SYSTEM Test_6 (* System Configuration *)
  (* Standard: 61499-1 *)
  (* Version 0.3, 2003-12-05, JHC, Rockwell Automation, Renamed from NEWSYSTEM. *)
  (* Version 0.2, 2002-11-05, JHC, Rockwell Automation, Fixed missing (empty) FBD in Application. *)
  (* Version 0.1, 2002-01-17, JHC, Rockwell Automation, Minor cleanup *)
  (* Version 0.0, 2000-05-27, JHC, Rockwell Automation *)
  APPLICATION APP1
  END_APPLICATION
  DEVICE DEV1 : FRAME_DEVICE(BOUNDS := [110,110,300,300], GRID := [1,1])
    RESOURCE RES1 : PANEL_RESOURCE(ROWS := 2, COLS := 2)
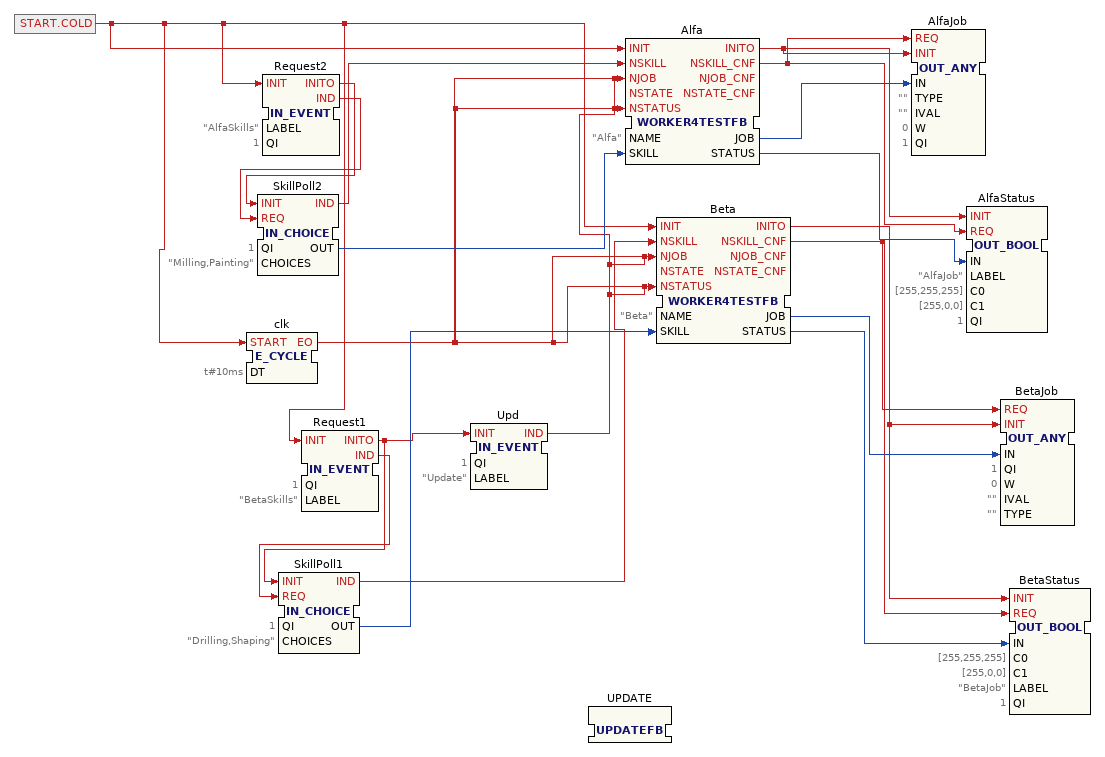
      FBS
        Alfa : WORKER4TESTFB(NAME := "Alfa");
        Beta : WORKER4TESTFB(NAME := "Beta");
        Request1 : IN_EVENT(QI := 1, LABEL := "BetaSkills");
        AlfaJob : OUT_ANY(TYPE := "", IVAL := "", W := 0, QI := 1);
        BetaJob : OUT_ANY(QI := 1, W := 0, IVAL := "", TYPE := "");
        AlfaStatus : OUT_BOOL(LABEL := "AlfaJob", C0 := [255,255,255], C1 := [255,0,0], QI := 1);
        BetaStatus : OUT_BOOL(C0 := [255,255,255], C1 := [255,0,0], LABEL := "BetaJob", QI := 1);
        UPDATE : UPDATEFB;
        clk : E_CYCLE(DT := t#10ms);
        SkillPoll1 : IN_CHOICE(QI := 1, CHOICES := "Drilling,Shaping");
        SkillPoll2 : IN_CHOICE(QI := 1, CHOICES := "Milling,Painting");
        Request2 : IN_EVENT(LABEL := "AlfaSkills", QI := 1);
        Upd : IN_EVENT(QI := 1, LABEL := "Update");
      END_FBS
      EVENT_CONNECTIONS
        START.COLD TO Alfa.INIT;
        START.COLD TO Beta.INIT;
        Alfa.NSKILL_CNF TO AlfaJob.REQ;
        Beta.NSKILL_CNF TO BetaJob.REQ;
        Beta.INITO TO BetaJob.INIT;
        Alfa.INITO TO AlfaJob.INIT;
        Alfa.INITO TO AlfaStatus.INIT;
        Alfa.NSKILL_CNF TO AlfaStatus.REQ;
        Beta.INITO TO BetaStatus.INIT;
        Beta.NSKILL_CNF TO BetaStatus.REQ;
        START.COLD TO clk.START;
        SkillPoll1.IND TO Beta.NSKILL;
        SkillPoll2.IND TO Alfa.NSKILL;
        Request1.INITO TO SkillPoll1.INIT;
        Request1.IND TO SkillPoll1.REQ;
        START.COLD TO Request1.INIT;
        START.COLD TO Request2.INIT;
        Request2.INITO TO SkillPoll2.INIT;
        Request2.IND TO SkillPoll2.REQ;
        clk.EO TO Alfa.NJOB;
        clk.EO TO Beta.NJOB;
        clk.EO TO Beta.NSTATUS;
        clk.EO TO Alfa.NSTATUS;
        Request1.INITO TO Upd.INIT;
        Upd.IND TO Beta.NJOB;
        Upd.IND TO Beta.NSTATUS;
        Upd.IND TO Alfa.NSTATUS;
        Upd.IND TO Alfa.NJOB;
      END_CONNECTIONS
      DATA_CONNECTIONS
        Beta.JOB TO BetaJob.IN;
        Alfa.JOB TO AlfaJob.IN;
        Alfa.STATUS TO AlfaStatus.IN;
        Beta.STATUS TO BetaStatus.IN;
        SkillPoll1.OUT TO Beta.SKILL;
        SkillPoll2.OUT TO Alfa.SKILL;
      END_CONNECTIONS
    END_RESOURCE
  END_DEVICE
END_SYSTEM
